// TIA Portal V19 export
TYPE "LAF_typeHeader"
// Information of the HMI header
// stored: Access Published
   STRUCT
      hmiToPlc { S7_SetPoint := 'True'} : "LAF_typeHeaderHmiToPlc";
      plcToHmi { S7_SetPoint := 'True'} : "LAF_typeHeaderPlcToHmi";
   END_STRUCT;
END_TYPE
